Fanuc KAREL source: SQRT.kl

PROGRAM T
%NOLOCKGROUP
VAR
 v0 : REAL
 res : REAL
BEGIN
 res = SQRT(v0)
END T
